Yaskawa INFORM job: STORMY.JBI

/JOB
//NAME STORMY
//POS
///NPOS 10,0,0,0
///TOOL 0
///PULSE
C000=-23851,23285,-36353,-11421,1798,9828
C001=-26011,19445,-29201,-8817,454,9184
C002=-26011,19445,-37457,-8145,-218,10248
C003=-19579,19445,-23825,-8145,6,7308
C004=-32299,19445,-29057,-9629,1070,6972
C005=-32299,19445,-34241,-9629,1070,6132
C006=-22603,18533,-33905,-7949,-1338,7560
C007=-27691,25397,-37217,-7949,-2738,5712
C008=-31099,29765,-35633,-7977,1546,5908
C009=-29515,27845,-37313,-4701,-1982,5152
//INST
///DATE 2014/10/12 15:50
///ATTR 0,0,0,0,0,0,0,0,0,0,0,0,0,1,0,0
///FRAME BASE
NOP
*Y
MOVJ C000 VJ=100.00 CONT
MOVJ C001 VJ=100.00 CONT
MOVJ C002 VJ=100.00 CONT
MOVJ C003 VJ=100.00 CONT
MOVJ C004 VJ=100.00 CONT
MOVJ C005 VJ=100.00 CONT
MOVJ C006 VJ=100.00 CONT
MOVJ C007 VJ=100.00 CONT
MOVJ C008 VJ=100.00 CONT
MOVJ C009 VJ=100.00 CONT
JUMP *Y
END
